(* Schneider Machine Expert - Basic project ProyekTrafficLight, file version 2.5.0.0 *)
(* ProjectInformations: Name=New project *)

HARDWARE
  Cpu 0: TM221CE24T
  EthernetConfiguration: NetworkName=M221, IpAllocationMode=FixedAddress, IpAddress=0.0.0.0, SubnetMask=0.0.0.0
  SerialLineConfiguration: Baud=Baud19200, Parity=ParityEven, DataBits=DataBits8, StopBits=StopBits1, PhysicalMedium=PhysicalMediumRs485, TransmissionMode=TransmissionModeModbusRtu, SlaveId=1, Addressing=SlaveAddressing
  MastTask: UsePeriodScanMode=false, PeriodScan=100
  FastTask: Period=255
  CpuBehavior: StartingMode=StartAsPreviousState, AutoSaveRamOnEeprom=true, WatchdogPeriod=250

SYMBOLS  (address, symbol, comment, settings)
  %TM0        [Type=TP, Base=OneSecond]
  %TM1        [Type=TP, Preset=1, Base=OneSecond]
  %C0         [Preset=14]
  %Q0.0     LAMPU_NYALA
  %Q0.2     HIJAU_1
  %Q0.3     KUNING_1

POU IO
  (* SectionNumber=1 *)

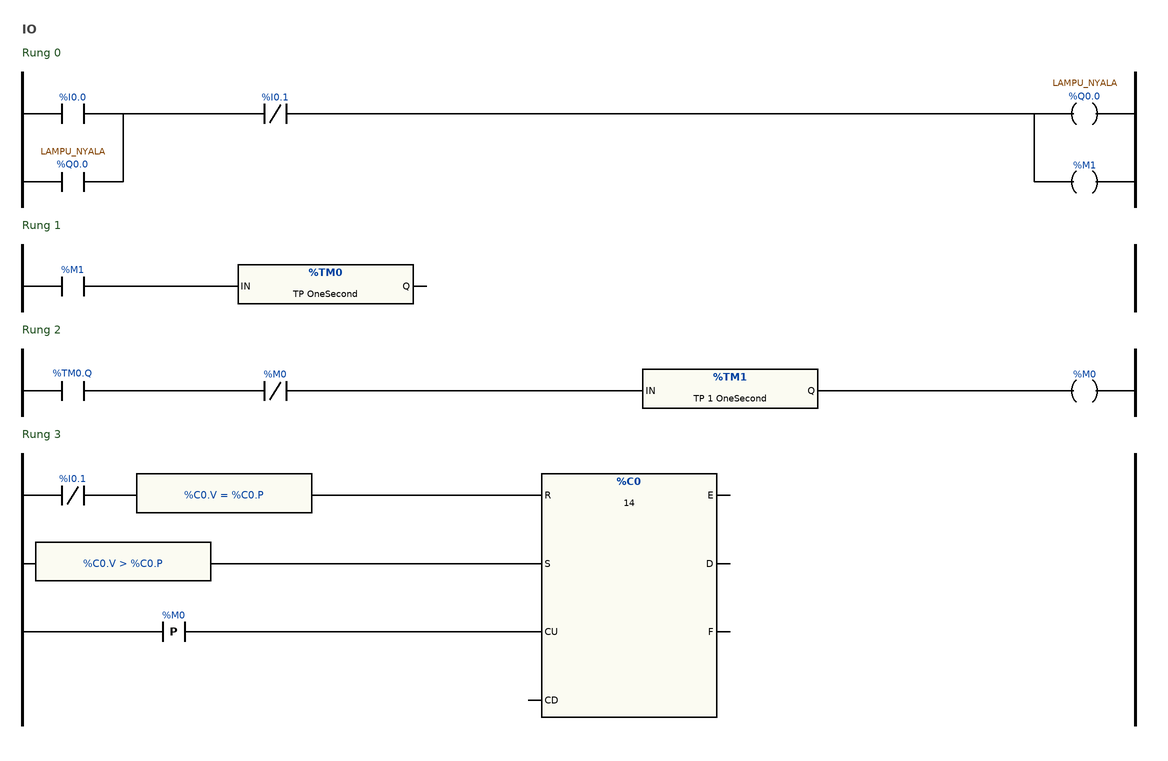

// Rung 0
  LD %I0.0
  OR %Q0.0                (* LAMPU_NYALA *)
  ANDN %I0.1
  ST %Q0.0                (* LAMPU_NYALA *)
  ST %M1
  // as ST:
  //   _t1 := (%I0.0 OR LAMPU_NYALA) AND NOT %I0.1;
  //   LAMPU_NYALA := _t1;
  //   %M1 := _t1;

// Rung 1
  BLK %TM0
  LD %M1
  IN
  END_BLK
  // as ST:
  //   %TM0(IN := %M1);

// Rung 2
  BLK %TM1
  LD %TM0.Q
  ANDN %M0
  IN
  OUT_BLK
  LD Q
  ST %M0
  END_BLK
  // as ST:
  //   %TM1(IN := %TM0.Q AND NOT %M0);
  //   %M0 := %TM1.Q;

// Rung 3
  BLK %C0
  LDN %I0.1
  AND [ %C0.V = %C0.P ]
  R
  LD [ %C0.V > %C0.P ]
  S
  LDR %M0
  CU
  END_BLK
  // as ST:
  //   %C0(R := NOT %I0.1 AND %C0.V = %C0.P, S := %C0.V > %C0.P, CU := RISING(%M0));

POU Lampu 1
  (* SectionNumber=2 *)

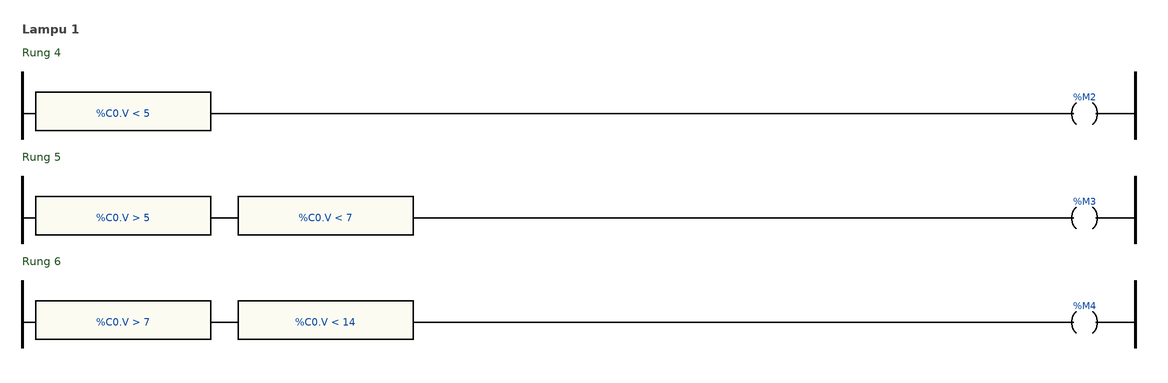

// Rung 4
  LD [ %C0.V < 5 ]
  ST %M2
  // as ST:
  //   %M2 := %C0.V < 5;

// Rung 5
  LD [ %C0.V > 5 ]
  AND [ %C0.V < 7 ]
  ST %M3
  // as ST:
  //   %M3 := %C0.V > 5 AND %C0.V < 7;

// Rung 6
  LD [ %C0.V > 7 ]
  AND [ %C0.V < 14 ]
  ST %M4
  // as ST:
  //   %M4 := %C0.V > 7 AND %C0.V < 14;

POU Lampu 2
  (* SectionNumber=3 *)

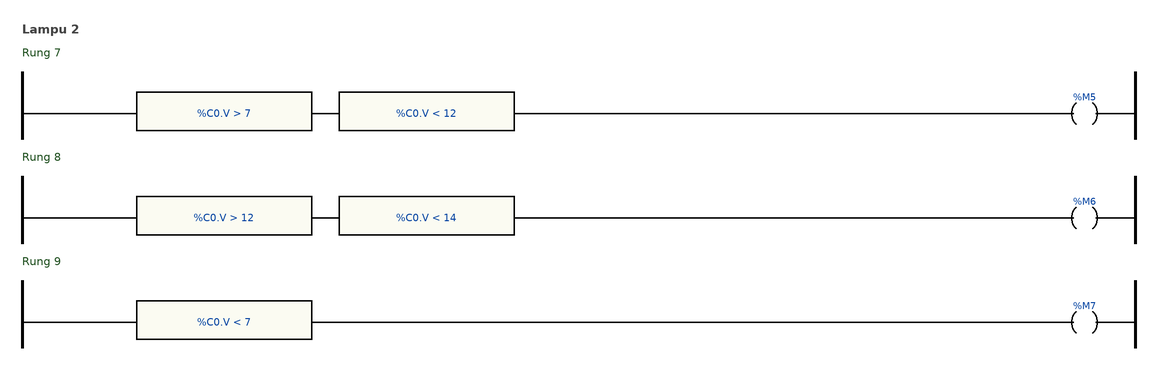

// Rung 7
  LD [ %C0.V > 7 ]
  AND [ %C0.V < 12 ]
  ST %M5
  // as ST:
  //   %M5 := %C0.V > 7 AND %C0.V < 12;

// Rung 8
  LD [ %C0.V > 12 ]
  AND [ %C0.V < 14 ]
  ST %M6
  // as ST:
  //   %M6 := %C0.V > 12 AND %C0.V < 14;

// Rung 9
  LD [ %C0.V < 7 ]
  ST %M7
  // as ST:
  //   %M7 := %C0.V < 7;
